// TIA Portal project "scl_2" (V18)

(* hardware
DEVICE "S7-1200 station_1"  S7-1200 Station
   slot 0: "Rack_0"  S7-1200 Rack  Rack  V1.0
   slot 1: "PLC_1"  CPU 1214C DC/DC/DC  6ES7 214-1AG40-0XB0  V4.6
*)

// ===== PLC "PLC_1"  CPU 1214C DC/DC/DC =====

VAR_GLOBAL   // PLC tag table "Default tag table"
   "START-STOP-1" AT %I0.0 : Bool;
   "START-STOP-2" AT %I0.1 : Bool;
   "MOTOR" AT %Q0.0 : Bool;
END_VAR

FUNCTION "Block_1" : Void   // FC1, SCL
{ S7_Optimized_Access := 'TRUE' }
VERSION : 0.1
BEGIN
   "MOTOR" := ("START-STOP-1" AND NOT "START-STOP-2") OR ("START-STOP-2" AND NOT "START-STOP-1");
END_FUNCTION

ORGANIZATION_BLOCK "Main"   // OB1, LAD, ProgramCycle
TITLE = "Main Program Sweep (Cycle)"
{ S7_Optimized_Access := 'TRUE' }
VERSION : 0.1
// SCL İLE MAİN AYNI ÇALIŞMA PRENSİBİNE SAHİP
   VAR_INPUT
      Initial_Call : Bool;   // Initial call of this OB
      Remanence : Bool;   // =True, if remanent data are available
   END_VAR
BEGIN

REGION Network 1
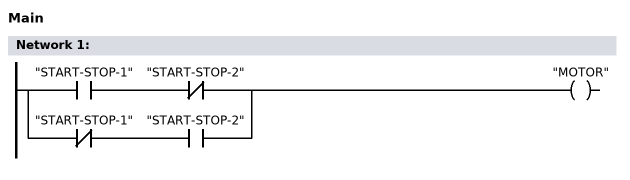
   RUNG wire#powerrail
      Contact( "START-STOP-1" )
      I_Contact( "START-STOP-2" )
      wire#w1
      Coil( "MOTOR" )
   END_RUNG
   RUNG wire#powerrail
      I_Contact( "START-STOP-1" )
      Contact( "START-STOP-2" )
   END_RUNG wire#w1
   // the same network as SCL:
   "MOTOR" := ("START-STOP-1" AND NOT "START-STOP-2") OR (NOT "START-STOP-1" AND "START-STOP-2");
END_REGION
END_ORGANIZATION_BLOCK